FUNCTION_BLOCK CapProviderCtrl (* Template for an empty basic function block *)
  (* Standard: 61499-2 *)
  (* Version 1.0, 2018-07-17, az *)
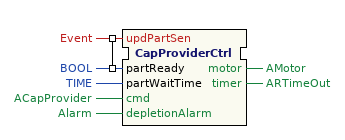
  EVENT_INPUT
    updPartSen WITH partReady;
  END_EVENT
  VAR_INPUT
    partReady : BOOL;
    partWaitTime : TIME;
  END_VAR
  SOCKETS
    cmd : ACapProvider;
    depletionAlarm : Alarm;
  END_SOCKETS
  PLUGS
    motor : AMotor;
    timer : ARTimeOut;
  END_PLUGS
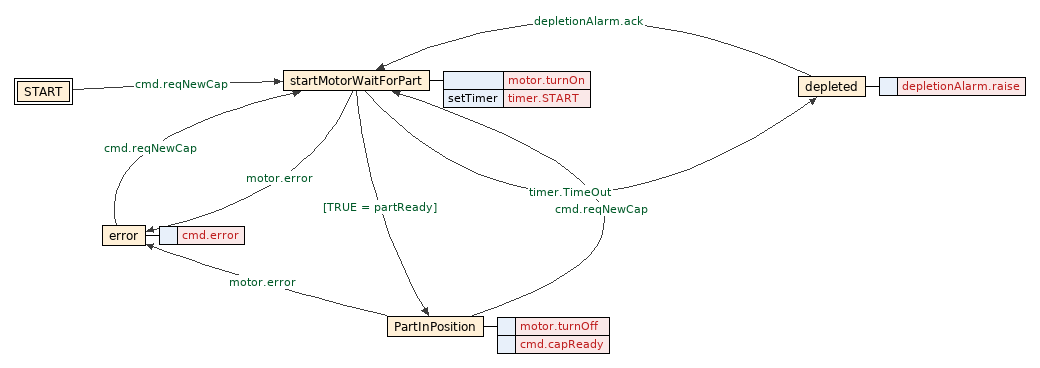
  EC_STATES
    START; (* Initial State *)
    error : -> cmd.error;
    startMotorWaitForPart : -> motor.turnOn, setTimer -> timer.START;
    PartInPosition : -> motor.turnOff, -> cmd.capReady;
    depleted : -> depletionAlarm.raise;
  END_STATES
  EC_TRANSITIONS
    START TO startMotorWaitForPart := cmd.reqNewCap;
    startMotorWaitForPart TO error := motor.error;
    error TO startMotorWaitForPart := cmd.reqNewCap;
    startMotorWaitForPart TO depleted := timer.TimeOut;
    depleted TO startMotorWaitForPart := depletionAlarm.ack;
    startMotorWaitForPart TO PartInPosition := [TRUE = partReady];
    PartInPosition TO error := motor.error;
    PartInPosition TO startMotorWaitForPart := cmd.reqNewCap;
  END_TRANSITIONS
  ALGORITHM setTimer IN ST: (* new algorithm *)
timer.DT := partWaitTime;
  END_ALGORITHM
END_FUNCTION_BLOCK
